// TIA Portal V19 export
FUNCTION_BLOCK "A0303_Spalla_FB"   // FB79, LAD
// stored: MemoryReserve 100, SetENOAutomatically false
   VAR_INPUT
      AreaInterface : "AreaInterface";
      ZSI : "udt_ZoneSafetyInterface";
      DSI : "udt_DeviceSafetyInterface";
      DataIn : Struct
         OP_Pos : Bool;
         FC_Aticoll_Paregg { ExternalWritable := 'False'} : Bool;
      END_STRUCT;
      CIn : Struct
         Manager : "Positioning_DOL_Machine_Manager";
         Antiribaltamento : Struct
            OutOfWorkspace : Bool;
         END_STRUCT;
         Pareggiatore : Struct
            ActualPosition : LReal;
         END_STRUCT;
      END_STRUCT;
      Config : Struct
         Ax : "Positioning_DOL_Machine_Config";
         DelayMissingCondition { ExternalAccessible := 'False'; ExternalVisible := 'False'; ExternalWritable := 'False'} : Time;
      END_STRUCT;
      HWID : Struct
         Ax_TEL1 : HW_SUBMODULE;
         Enc_IO : HW_SUBMODULE;
      END_STRUCT;
   END_VAR
   VAR_OUTPUT
      MachineInterface { ExternalAccessible := 'False'; ExternalVisible := 'False'; ExternalWritable := 'False'} : "MachineInterface";
      COut : Struct
         Ax : "Positioning_DOL_Machine_COut";
      END_STRUCT;
   END_VAR
   VAR_IN_OUT
      Par : Struct
         Ax : "Positioning_DOL_Machine_Par";
         Ax_Pers : "Positioning_DOL_Machine_Pers_Data";
         Enc : "PosFbk_RTN";
      END_STRUCT;
      Par_Mach : Struct
         MinDistanzaConParegg : LReal;
         ToleranceWindow : LReal;
      END_STRUCT;
   END_VAR
   VAR
      Alarm : Struct
         Ax : "Positioning_DOL_Machine_Alr";
         Enc : "PosFbk_Encoder_Alr";
      END_STRUCT;
      Warning : Struct
         Ax : "Positioning_DOL_Machine_Wng";
         SW_Limit_AntiCollision : Bool;
         OP_POS_MissingCnd : Bool;   // Mancanza comando arresto
      END_STRUCT;
      HMI : Struct
         PbPreset : Bool;
         B_Preset_UM2 : Bool;
         PresetValue : LReal;
      END_STRUCT;
      Sts : Struct
         AlarmsPresence : Bool;
         WarningsPresence : Bool;
         OP_CanMoveFreely : Bool;
         OP_Pos_Cnd : Bool;
      END_STRUCT;
      Ctrl : Struct
         OP_Pos_Aut : Bool;
         OP_Pos_Run : Bool;
         OP_Pos_Man : Bool;
         OP_Pos : Bool;
      END_STRUCT;
      Ax : "Positioning_DOL_Machine_FB";
      Enc : "PosFbk_SickAFM60";
      Enc_ITF : "PosFbk_ITF";
      AUX { ExternalAccessible := 'False'; ExternalVisible := 'False'; ExternalWritable := 'False'} : Struct
         OP_Pos_PB : Bool;
      END_STRUCT;
      TON_OP_POS_MissingCnd : IEC_TIMER;
      TON_DistanzaOK : IEC_TIMER;
   END_VAR
   VAR_TEMP
      PE : Struct
         OP_Pos_PB : Bool;
      END_STRUCT;
      ActualDifference : LReal;
   END_VAR
   VAR_TEMP   // added for the SCL form of the ladder/FBD networks
      _w1 : Bool;
   END_VAR
BEGIN

REGION Network 1: Operazione può muoversi liberamente perchè non sposta nessun BEAM
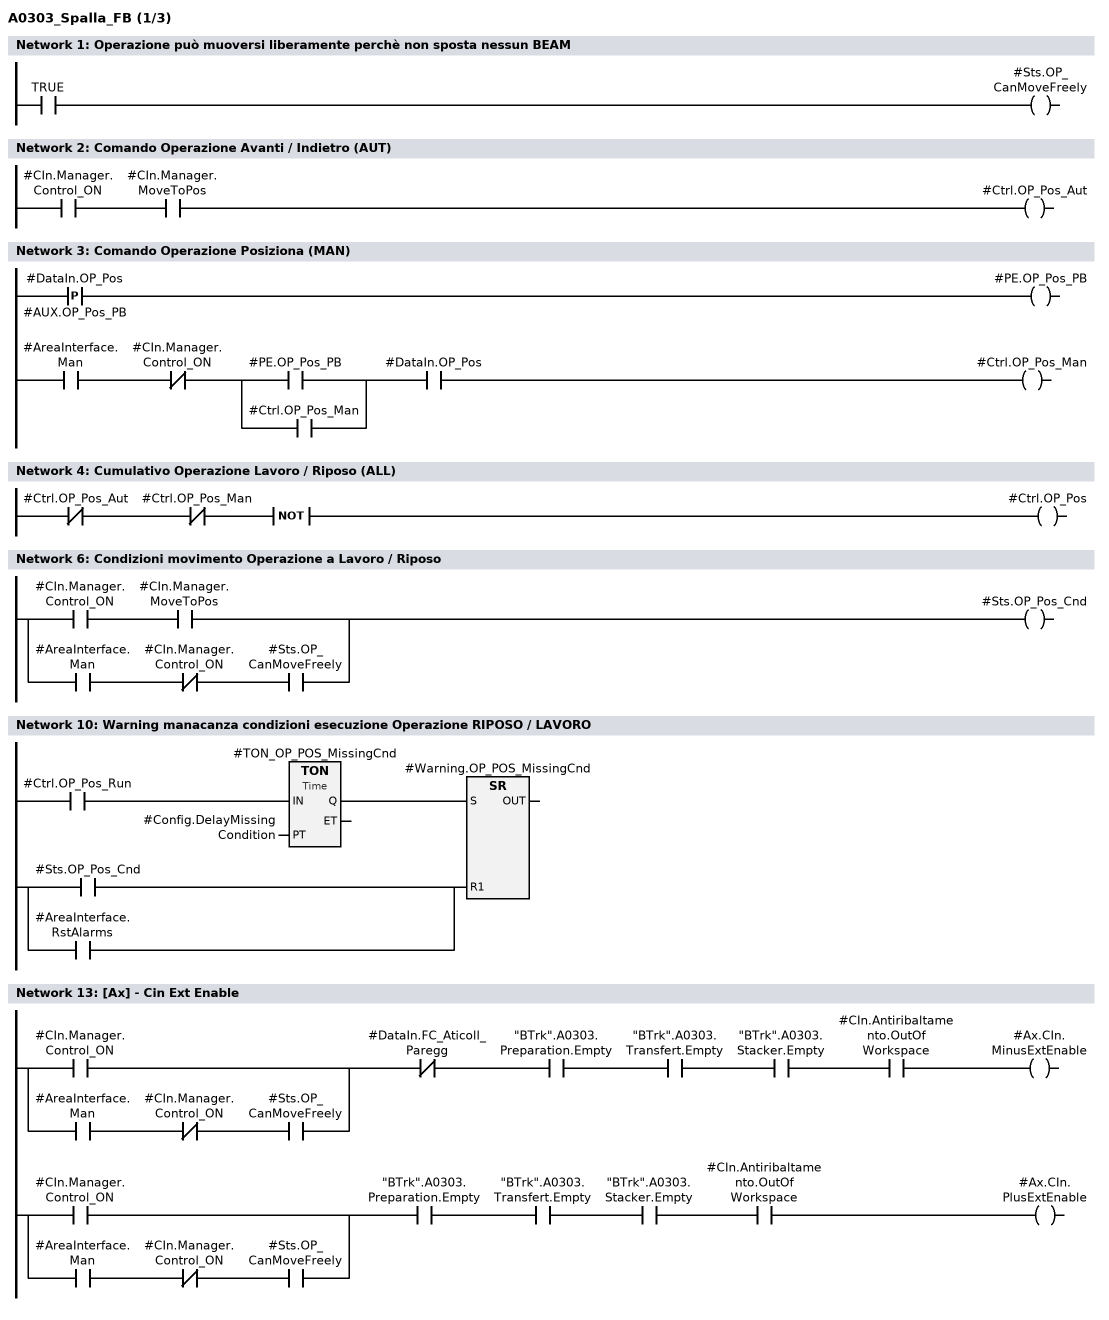
   RUNG wire#powerrail
      Contact( TRUE )
      Coil( #Sts.OP_CanMoveFreely )
   END_RUNG
   // the same network as SCL:
   #Sts.OP_CanMoveFreely := TRUE;
END_REGION

REGION Network 2: Comando Operazione Avanti / Indietro (AUT)
   RUNG wire#powerrail
      Contact( #CIn.Manager.Control_ON )
      Contact( #CIn.Manager.MoveToPos )
      Coil( #Ctrl.OP_Pos_Aut )
   END_RUNG
   // the same network as SCL:
   #Ctrl.OP_Pos_Aut := #CIn.Manager.Control_ON AND #CIn.Manager.MoveToPos;
END_REGION

REGION Network 3: Comando Operazione Posiziona (MAN)
   RUNG wire#powerrail
      P_Contact(operand := #DataIn.OP_Pos, bit := #AUX.OP_Pos_PB)
      Coil( #PE.OP_Pos_PB )
   END_RUNG
   RUNG wire#powerrail
      Contact( #AreaInterface.Man )
      I_Contact( #CIn.Manager.Control_ON )
      wire#w1
      Contact( #PE.OP_Pos_PB )
      wire#w2
      Contact( #DataIn.OP_Pos )
      Coil( #Ctrl.OP_Pos_Man )
   END_RUNG
   RUNG wire#w1
      Contact( #Ctrl.OP_Pos_Man )
   END_RUNG wire#w2
   // the same network as SCL:
   #_w1 := #DataIn.OP_Pos AND NOT #AUX.OP_Pos_PB;   // rising edge of #DataIn.OP_Pos
   #AUX.OP_Pos_PB := #DataIn.OP_Pos;
   #PE.OP_Pos_PB := #_w1;
   #Ctrl.OP_Pos_Man := #AreaInterface.Man AND NOT #CIn.Manager.Control_ON AND (#PE.OP_Pos_PB OR #Ctrl.OP_Pos_Man) AND #DataIn.OP_Pos;
END_REGION

REGION Network 4: Cumulativo Operazione Lavoro / Riposo (ALL)
   RUNG wire#powerrail
      I_Contact( #Ctrl.OP_Pos_Aut )
      I_Contact( #Ctrl.OP_Pos_Man )
      Not()
      Coil( #Ctrl.OP_Pos )
   END_RUNG
   // the same network as SCL:
   #Ctrl.OP_Pos := NOT (NOT #Ctrl.OP_Pos_Aut AND NOT #Ctrl.OP_Pos_Man);
END_REGION

REGION Network 5: <+>
END_REGION

REGION Network 6: Condizioni movimento Operazione a Lavoro / Riposo
   RUNG wire#powerrail
      Contact( #CIn.Manager.Control_ON )
      Contact( #CIn.Manager.MoveToPos )
      wire#w1
      Coil( #Sts.OP_Pos_Cnd )
   END_RUNG
   RUNG wire#powerrail
      Contact( #AreaInterface.Man )
      I_Contact( #CIn.Manager.Control_ON )
      Contact( #Sts.OP_CanMoveFreely )
   END_RUNG wire#w1
   // the same network as SCL:
   #Sts.OP_Pos_Cnd := (#CIn.Manager.Control_ON AND #CIn.Manager.MoveToPos) OR (#AreaInterface.Man AND NOT #CIn.Manager.Control_ON AND #Sts.OP_CanMoveFreely);
END_REGION

REGION Network 7 (SCL): Cin Manager Comando posizionamento
   // CIn Manager  Control ON se ho un richiesta di comando attiva
   #Ax.CIn.Manager.Control_ON := #Ctrl.OP_Pos;
   #Ax.CIn.Manager.Speed := #CIn.Manager.Speed;

   // Resetto i comandi se non c'è nessuna richiesta attiva
   IF NOT #Ax.CIn.Manager.Control_ON THEN
       #Ax.CIn.Manager.MoveToPos := FALSE;
   END_IF;

   IF #Ctrl.OP_Pos AND #Sts.OP_Pos_Cnd THEN
       //In posizione di attrezzaggio
       //
       #Ax.CIn.Manager.MoveToPos := #CIn.Manager.MoveToPos;
       #Ax.CIn.Manager.Pos := #CIn.Manager.Pos;
   ELSE
       #Ax.CIn.Manager.MoveToPos := FALSE;
   END_IF;
END_REGION

REGION Network 8 (SCL): CIn Abilitazioni Stop Manager
   // CIn Manager Stop per richiesta apertura safety
   // 
   #Ax.CIn.Manager.EnableStopDoorOpeningReq := #CIn.Manager.EnableStopDoorOpeningReq;

   // CIn Manager Stop in fase delle macchine precedenti
   // 
   #Ax.CIn.Manager.EnableStopInPhase := #CIn.Manager.EnableStopInPhase;

   // CIn Manager Stop programmato configurabile a piacere
   // 
   #Ax.CIn.Manager.EnableStopProgrammed := #CIn.Manager.EnableStopProgrammed;
END_REGION

REGION Network 9: <+>
END_REGION

REGION Network 10: Warning manacanza condizioni esecuzione Operazione RIPOSO / LAVORO
   RUNG wire#powerrail
      Contact( #Ctrl.OP_Pos_Run )
      { S7_Templates := "time_type := Time" } #TON_OP_POS_MissingCnd.TON(pt := #Config.DelayMissingCondition, et =>)
      S_SR(operand := #Warning.OP_POS_MissingCnd, r1 := wire#w1)
   END_RUNG
   RUNG wire#powerrail
      Contact( #Sts.OP_Pos_Cnd )
   END_RUNG wire#w1
   RUNG wire#powerrail
      Contact( #AreaInterface.RstAlarms )
   END_RUNG wire#w1
   // the same network as SCL:
   #TON_OP_POS_MissingCnd.TON(IN := #Ctrl.OP_Pos_Run, PT := #Config.DelayMissingCondition);
   IF #TON_OP_POS_MissingCnd.Q THEN
       #Warning.OP_POS_MissingCnd := TRUE;   // SR flip-flop
   END_IF;
   IF #Sts.OP_Pos_Cnd OR #AreaInterface.RstAlarms THEN #Warning.OP_POS_MissingCnd := FALSE; END_IF;
END_REGION

REGION Network 11: <+>
END_REGION

REGION Network 12: <<< SPALLA>>>
END_REGION

REGION Network 13: [Ax] - Cin Ext Enable
   RUNG wire#powerrail
      Contact( #CIn.Manager.Control_ON )
      wire#w1
      I_Contact( #DataIn.FC_Aticoll_Paregg )
      Contact( "BTrk".A0303.Preparation.Empty )
      Contact( "BTrk".A0303.Transfert.Empty )
      Contact( "BTrk".A0303.Stacker.Empty )
      Contact( #CIn.Antiribaltamento.OutOfWorkspace )
      Coil( #Ax.CIn.MinusExtEnable )
   END_RUNG
   RUNG wire#powerrail
      Contact( #AreaInterface.Man )
      I_Contact( #CIn.Manager.Control_ON )
      Contact( #Sts.OP_CanMoveFreely )
   END_RUNG wire#w1
   RUNG wire#powerrail
      Contact( #CIn.Manager.Control_ON )
      wire#w2
      Contact( "BTrk".A0303.Preparation.Empty )
      Contact( "BTrk".A0303.Transfert.Empty )
      Contact( "BTrk".A0303.Stacker.Empty )
      Contact( #CIn.Antiribaltamento.OutOfWorkspace )
      Coil( #Ax.CIn.PlusExtEnable )
   END_RUNG
   RUNG wire#powerrail
      Contact( #AreaInterface.Man )
      I_Contact( #CIn.Manager.Control_ON )
      Contact( #Sts.OP_CanMoveFreely )
   END_RUNG wire#w2
   // the same network as SCL:
   #Ax.CIn.MinusExtEnable := (#CIn.Manager.Control_ON OR (#AreaInterface.Man AND NOT #CIn.Manager.Control_ON AND #Sts.OP_CanMoveFreely)) AND NOT #DataIn.FC_Aticoll_Paregg AND "BTrk".A0303.Preparation.Empty AND "BTrk".A0303.Transfert.Empty AND "BTrk".A0303.Stacker.Empty AND #CIn.Antiribaltamento.OutOfWorkspace;
   #Ax.CIn.PlusExtEnable := (#CIn.Manager.Control_ON OR (#AreaInterface.Man AND NOT #CIn.Manager.Control_ON AND #Sts.OP_CanMoveFreely)) AND "BTrk".A0303.Preparation.Empty AND "BTrk".A0303.Transfert.Empty AND "BTrk".A0303.Stacker.Empty AND #CIn.Antiribaltamento.OutOfWorkspace;
END_REGION

REGION Network 14: [Ax] - CIn External alarm
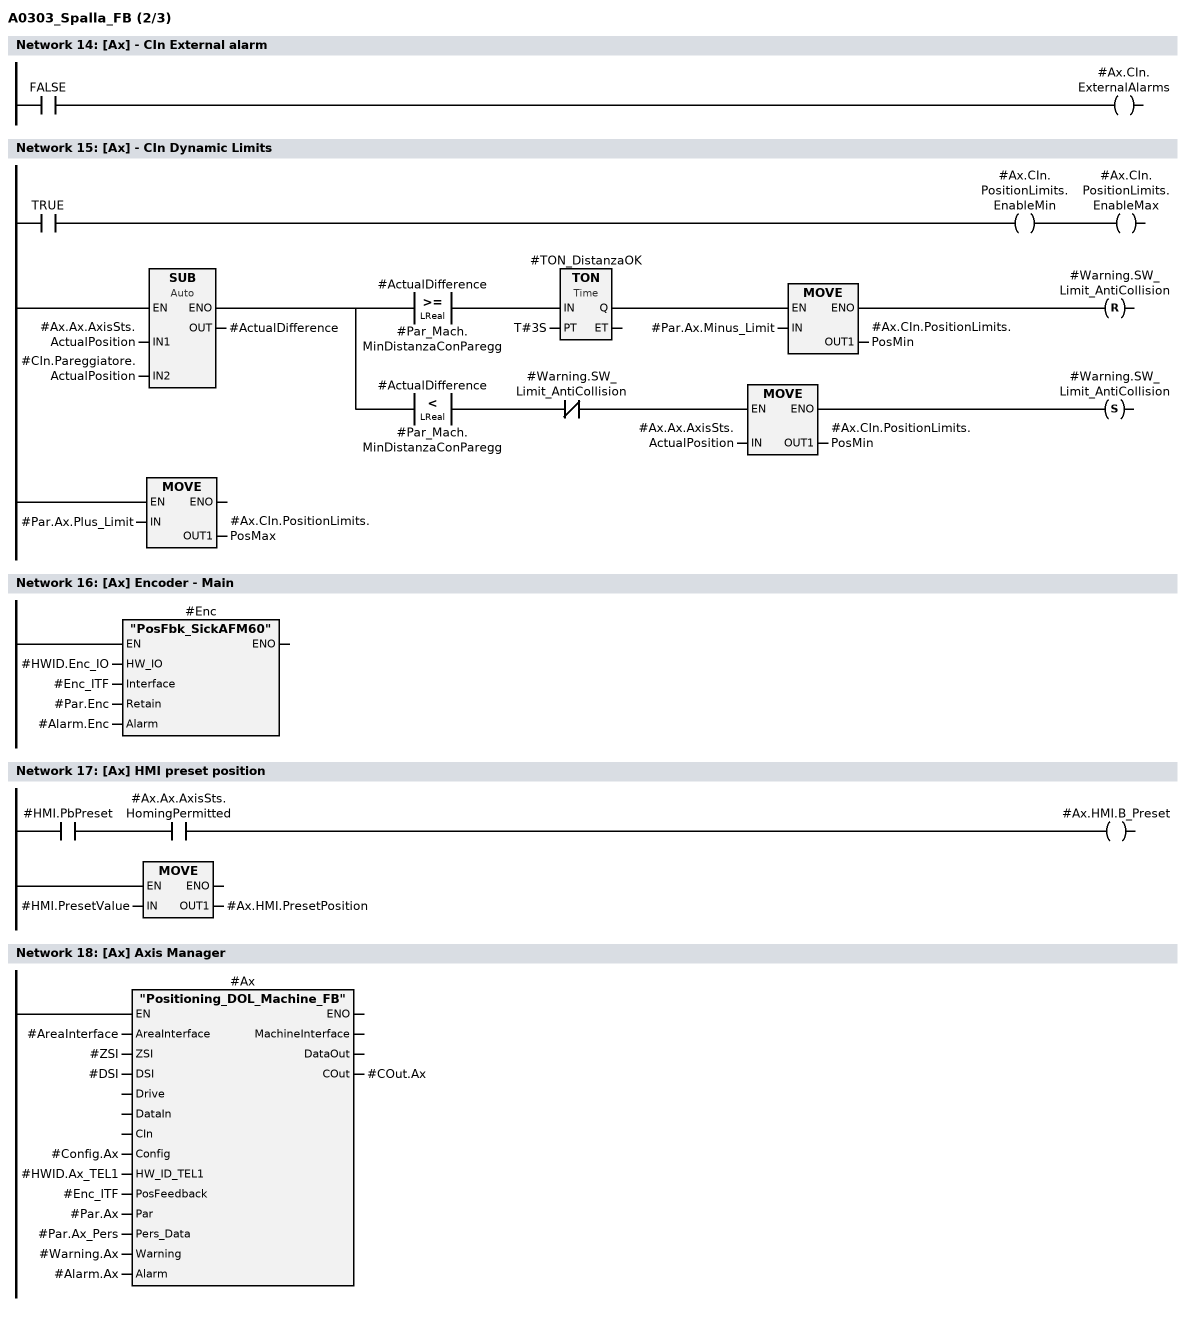
   RUNG wire#powerrail
      Contact( FALSE )
      Coil( #Ax.CIn.ExternalAlarms )
   END_RUNG
   // the same network as SCL:
   #Ax.CIn.ExternalAlarms := FALSE;
END_REGION

REGION Network 15: [Ax] - CIn Dynamic Limits
   RUNG wire#powerrail
      Contact( TRUE )
      Coil( #Ax.CIn.PositionLimits.EnableMin )
      Coil( #Ax.CIn.PositionLimits.EnableMax )
   END_RUNG
   RUNG wire#powerrail
      Sub(in1 := #Ax.Ax.AxisSts.ActualPosition, in2 := #CIn.Pareggiatore.ActualPosition, out => #ActualDifference)
      wire#w1
      { S7_Templates := "SrcType := LReal" } GE_Contact(in1 := #ActualDifference, in2 := #Par_Mach.MinDistanzaConParegg)
      { S7_Templates := "time_type := Time" } #TON_DistanzaOK.TON(pt := T#3S, et =>)
      Move(in := #Par.Ax.Minus_Limit, out1 => #Ax.CIn.PositionLimits.PosMin)
      R_Coil( #Warning.SW_Limit_AntiCollision )
   END_RUNG
   RUNG wire#w1
      { S7_Templates := "SrcType := LReal" } LT_Contact(in1 := #ActualDifference, in2 := #Par_Mach.MinDistanzaConParegg)
      I_Contact( #Warning.SW_Limit_AntiCollision )
      Move(in := #Ax.Ax.AxisSts.ActualPosition, out1 => #Ax.CIn.PositionLimits.PosMin)
      S_Coil( #Warning.SW_Limit_AntiCollision )
   END_RUNG
   RUNG wire#powerrail
      Move(in := #Par.Ax.Plus_Limit, out1 => #Ax.CIn.PositionLimits.PosMax)
   END_RUNG
   // the same network as SCL:
   #Ax.CIn.PositionLimits.EnableMin := TRUE;
   #Ax.CIn.PositionLimits.EnableMax := TRUE;
   #ActualDifference := #Ax.Ax.AxisSts.ActualPosition - #CIn.Pareggiatore.ActualPosition;
   #TON_DistanzaOK.TON(IN := #ActualDifference >= #Par_Mach.MinDistanzaConParegg, PT := T#3S);
   IF #TON_DistanzaOK.Q THEN
       #Ax.CIn.PositionLimits.PosMin := #Par.Ax.Minus_Limit;
       #Warning.SW_Limit_AntiCollision := FALSE;
   END_IF;
   IF (#ActualDifference < #Par_Mach.MinDistanzaConParegg) AND NOT #Warning.SW_Limit_AntiCollision THEN
       #Ax.CIn.PositionLimits.PosMin := #Ax.Ax.AxisSts.ActualPosition;
       #Warning.SW_Limit_AntiCollision := TRUE;
   END_IF;
   #Ax.CIn.PositionLimits.PosMax := #Par.Ax.Plus_Limit;
END_REGION

REGION Network 16: [Ax] Encoder - Main
   RUNG wire#powerrail
      #Enc(HW_IO := #HWID.Enc_IO, Interface := #Enc_ITF, Retain := #Par.Enc, Alarm := #Alarm.Enc)
   END_RUNG
   // the same network as SCL:
   #Enc(HW_IO := #HWID.Enc_IO, Interface := #Enc_ITF, Retain := #Par.Enc, Alarm := #Alarm.Enc);   // "PosFbk_SickAFM60"
END_REGION

REGION Network 17: [Ax] HMI preset position
   RUNG wire#powerrail
      Contact( #HMI.PbPreset )
      Contact( #Ax.Ax.AxisSts.HomingPermitted )
      Coil( #Ax.HMI.B_Preset )
   END_RUNG
   RUNG wire#powerrail
      Move(in := #HMI.PresetValue, out1 => #Ax.HMI.PresetPosition)
   END_RUNG
   // the same network as SCL:
   #Ax.HMI.B_Preset := #HMI.PbPreset AND #Ax.Ax.AxisSts.HomingPermitted;
   #Ax.HMI.PresetPosition := #HMI.PresetValue;
END_REGION

REGION Network 18: [Ax] Axis Manager
   RUNG wire#powerrail
      #Ax(AreaInterface := #AreaInterface, ZSI := #ZSI, DSI := #DSI, Drive :=, DataIn :=, CIn :=, Config := #Config.Ax, HW_ID_TEL1 := #HWID.Ax_TEL1, PosFeedback := #Enc_ITF, Par := #Par.Ax, Pers_Data := #Par.Ax_Pers, Warning := #Warning.Ax, Alarm := #Alarm.Ax, MachineInterface =>, DataOut =>, COut => #COut.Ax)
   END_RUNG
   // the same network as SCL:
   #Ax(AreaInterface := #AreaInterface,   // "Positioning_DOL_Machine_FB"
       ZSI := #ZSI,
       DSI := #DSI,
       Config := #Config.Ax,
       HW_ID_TEL1 := #HWID.Ax_TEL1,
       PosFeedback := #Enc_ITF,
       Par := #Par.Ax,
       Pers_Data := #Par.Ax_Pers,
       Warning := #Warning.Ax,
       Alarm := #Alarm.Ax,
       COut => #COut.Ax);
END_REGION

REGION Network 20: <+>
END_REGION

REGION Network 21: <<< MACHINE STATUS >>>
END_REGION

REGION Network 22: Collect machine to zone interface
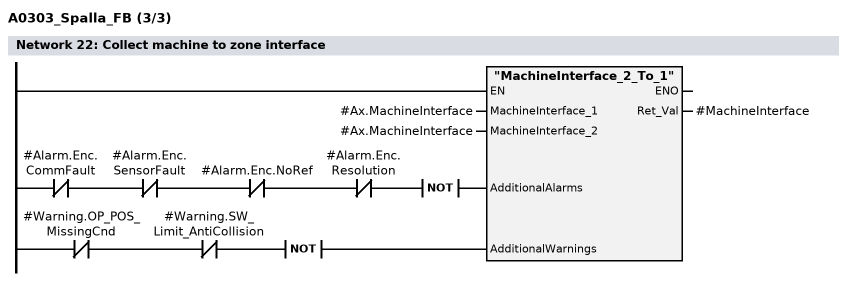
   RUNG wire#powerrail
      "MachineInterface_2_To_1"(AdditionalAlarms := wire#w1, AdditionalWarnings := wire#w2, MachineInterface_1 := #Ax.MachineInterface, MachineInterface_2 := #Ax.MachineInterface, Ret_Val => #MachineInterface)
   END_RUNG
   RUNG wire#powerrail
      I_Contact( #Alarm.Enc.CommFault )
      I_Contact( #Alarm.Enc.SensorFault )
      I_Contact( #Alarm.Enc.NoRef )
      I_Contact( #Alarm.Enc.Resolution )
      Not()
   END_RUNG wire#w1
   RUNG wire#powerrail
      I_Contact( #Warning.OP_POS_MissingCnd )
      I_Contact( #Warning.SW_Limit_AntiCollision )
      Not()
   END_RUNG wire#w2
   // the same network as SCL:
   #MachineInterface := "MachineInterface_2_To_1"(MachineInterface_1 := #Ax.MachineInterface,
                           MachineInterface_2 := #Ax.MachineInterface,
                           AdditionalAlarms := NOT (NOT #Alarm.Enc.CommFault AND NOT #Alarm.Enc.SensorFault AND NOT #Alarm.Enc.NoRef AND NOT #Alarm.Enc.Resolution),
                           AdditionalWarnings := NOT (NOT #Warning.OP_POS_MissingCnd AND NOT #Warning.SW_Limit_AntiCollision));
END_REGION
END_FUNCTION_BLOCK
